% RSLogix 500 project second_Version.RSS, saved by version 8.30.00.16 %
PROJECT "UNTITLED"    % processor: Bul.1763 MicroLogix 1100 Series B %

PROGRAM FILES
  LAD 2   5 rungs
  LAD 3 "CYCLE"  6 rungs
  LAD 4 "ALARMS"  9 rungs
  LAD 5 "IO"  13 rungs
  LAD 6 "LOGIC"  5 rungs

DATA FILES
  O0 OUTPUT  4 elements
  I1 INPUT  6 elements
  S2 STATUS  66 elements
  B3 BINARY  6 elements
  T4 TIMER  4 elements
  C5 COUNTER  1 elements
  R6 CONTROL  1 elements
  N7 INTEGER  4 elements
  F8 FLOAT  1 elements

LADDER 2
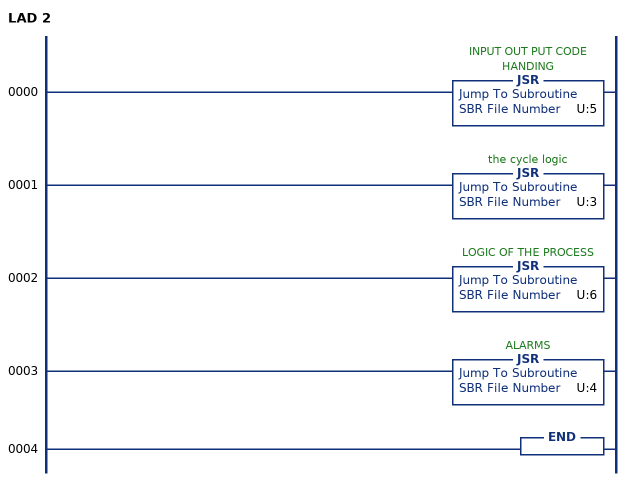
% Rung: 0 %
SOR JSR U:5 EOR
%   U:5  "INPUT OUT PUT CODE HANDING" %
% Rung: 1 %
SOR JSR U:3 EOR
%   U:3  "the cycle logic" %
% Rung: 2 %
SOR JSR U:6 EOR
%   U:6  "LOGIC OF THE PROCESS" %
% Rung: 3 %
SOR JSR U:4 EOR
%   U:4  "ALARMS" %
% Rung: 4 %
SOR END EOR

LADDER 3 "CYCLE"
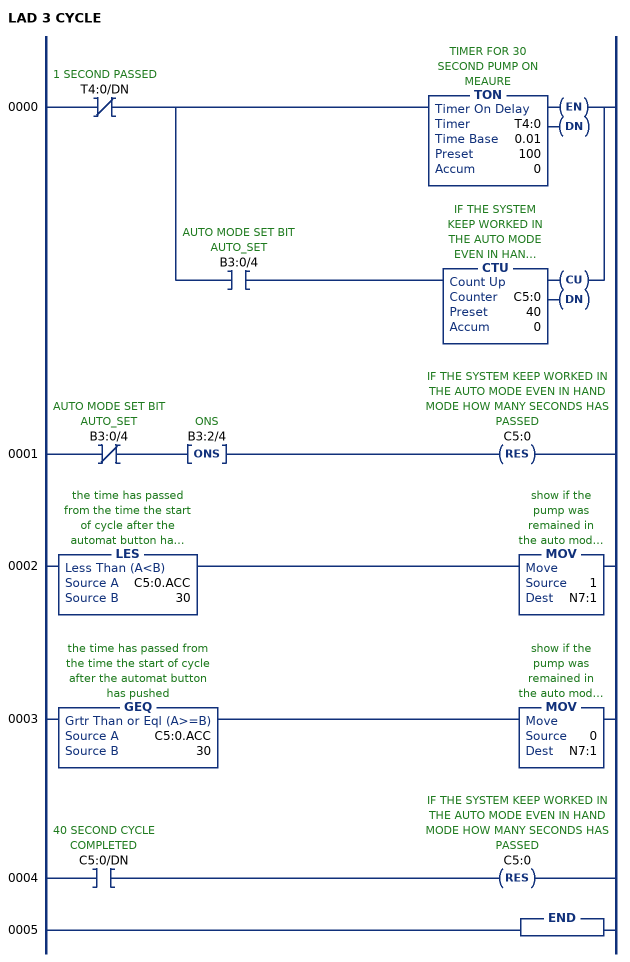
% Rung: 0 %
SOR XIO T4:0/DN BST TON T4:0 0.01 100 0 NXB XIC B3:0/4 CTU C5:0 40 0 BND EOR
%   T4:0/DN  "1 SECOND PASSED" %
%   T4:0  "TIMER FOR 30 SECOND PUMP ON MEAURE" %
%   B3:0/4  AUTO_SET  "AUTO MODE SET BIT" %
%   C5:0  "IF THE SYSTEM KEEP WORKED IN THE AUTO MODE EVEN IN HAND MODE HOW MANY SECONDS HAS PASSED" %
% Rung: 1 %
SOR XIO B3:0/4 ONS B3:2/4 RES C5:0 EOR
%   B3:0/4  AUTO_SET  "AUTO MODE SET BIT" %
%   B3:2/4  "ONS" %
%   C5:0  "IF THE SYSTEM KEEP WORKED IN THE AUTO MODE EVEN IN HAND MODE HOW MANY SECONDS HAS PASSED" %
% Rung: 2 %
SOR LES C5:0.ACC 30 MOV 1 N7:1 EOR
%   C5:0.ACC  "the time has passed from the time the start of cycle after the automat button has pushed" %
%   N7:1  MODE_REF  "show if the pump was remained in the auto mode it should be on which part 1= on mode 0 = off" %
% Rung: 3 %
SOR GEQ C5:0.ACC 30 MOV 0 N7:1 EOR
%   C5:0.ACC  "the time has passed from the time the start of cycle after the automat button has pushed" %
%   N7:1  MODE_REF  "show if the pump was remained in the auto mode it should be on which part 1= on mode 0 = off" %
% Rung: 4 %
SOR XIC C5:0/DN RES C5:0 EOR
%   C5:0/DN  "40 SECOND CYCLE COMPLETED" %
%   C5:0  "IF THE SYSTEM KEEP WORKED IN THE AUTO MODE EVEN IN HAND MODE HOW MANY SECONDS HAS PASSED" %
% Rung: 5 %
SOR END EOR

LADDER 4 "ALARMS"
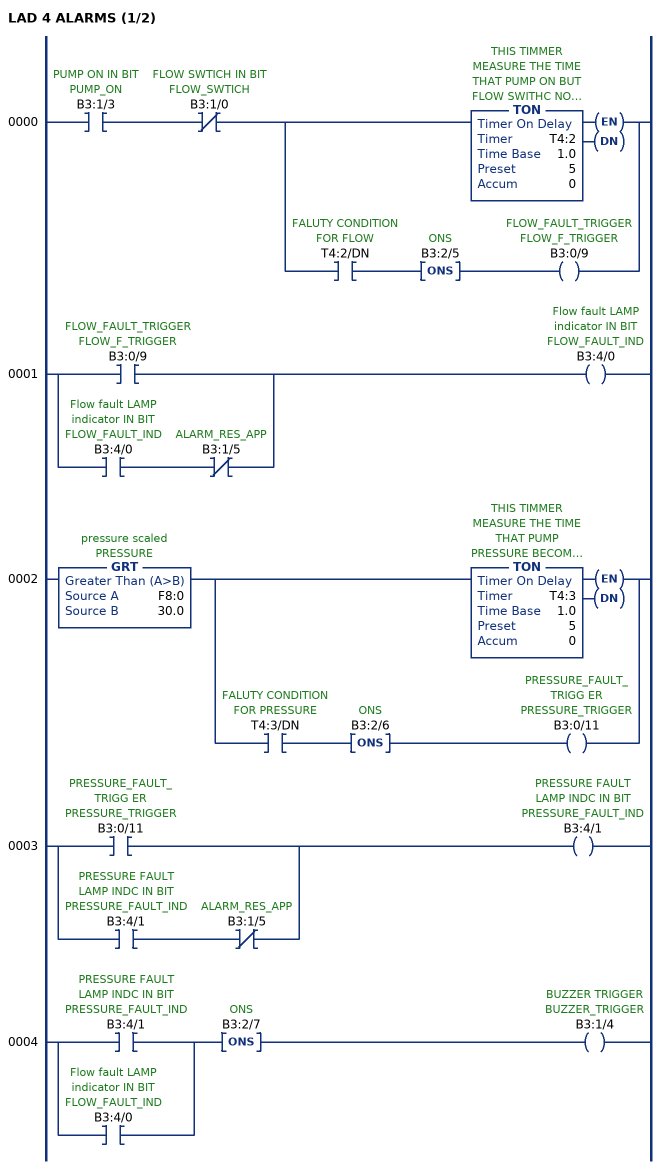
% Rung: 0 %
SOR XIC B3:1/3 XIO B3:1/0 BST TON T4:2 1.0 5 0 NXB XIC T4:2/DN ONS B3:2/5 OTE B3:0/9 BND EOR
%   B3:1/3  PUMP_ON  "PUMP ON IN BIT" %
%   B3:1/0  FLOW_SWTICH  "FLOW SWTICH IN BIT" %
%   T4:2  FLOW_AL_TIM  "THIS TIMMER MEASURE THE TIME THAT PUMP ON BUT FLOW SWITHC NOT TURN ON" %
%   T4:2/DN  "FALUTY CONDITION FOR FLOW" %
%   B3:2/5  "ONS" %
%   B3:0/9  FLOW_F_TRIGGER  "FLOW_FAULT_TRIGGER" %
% Rung: 1 %
SOR BST XIC B3:0/9 NXB XIC B3:4/0 XIO B3:1/5 BND OTE B3:4/0 EOR
%   B3:0/9  FLOW_F_TRIGGER  "FLOW_FAULT_TRIGGER" %
%   B3:4/0  FLOW_FAULT_IND  "Flow fault LAMP indicator IN BIT" %
%   B3:1/5  ALARM_RES_APP %
% Rung: 2 %
SOR GRT F8:0 30.0 BST TON T4:3 1.0 5 0 NXB XIC T4:3/DN ONS B3:2/6 OTE B3:0/11 BND EOR
%   F8:0  PRESSURE  "pressure scaled" %
%   T4:3  PRESSURE_AL_TIM  "THIS TIMMER MEASURE THE TIME THAT PUMP PRESSURE BECOME MORE THAN 30 PSI" %
%   T4:3/DN  "FALUTY CONDITION FOR PRESSURE" %
%   B3:2/6  "ONS" %
%   B3:0/11  PRESSURE_TRIGGER  "PRESSURE_FAULT_TRIGG ER" %
% Rung: 3 %
SOR BST XIC B3:0/11 NXB XIC B3:4/1 XIO B3:1/5 BND OTE B3:4/1 EOR
%   B3:0/11  PRESSURE_TRIGGER  "PRESSURE_FAULT_TRIGG ER" %
%   B3:4/1  PRESSURE_FAULT_IND  "PRESSURE FAULT LAMP INDC IN BIT" %
%   B3:1/5  ALARM_RES_APP %
% Rung: 4 %
SOR BST XIC B3:4/1 NXB XIC B3:4/0 BND ONS B3:2/7 OTE B3:1/4 EOR
%   B3:4/1  PRESSURE_FAULT_IND  "PRESSURE FAULT LAMP INDC IN BIT" %
%   B3:4/0  FLOW_FAULT_IND  "Flow fault LAMP indicator IN BIT" %
%   B3:2/7  "ONS" %
%   B3:1/4  BUZZER_TRIGGER  "BUZZER TRIGGER" %

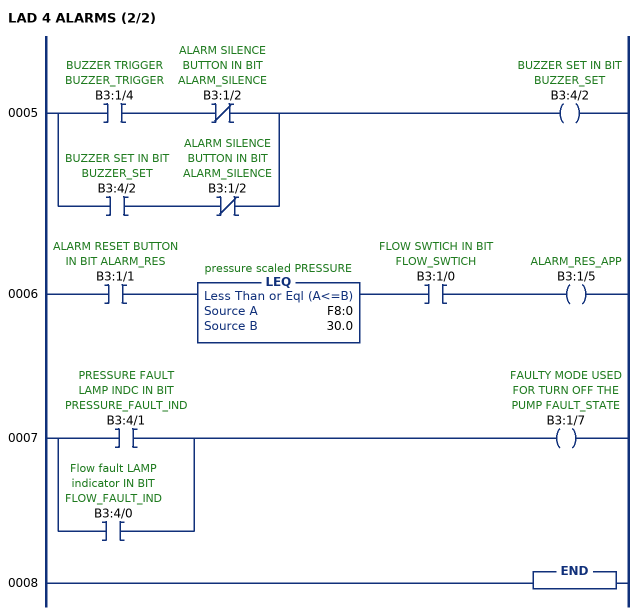
% Rung: 5 %
SOR BST XIC B3:1/4 XIO B3:1/2 NXB XIC B3:4/2 XIO B3:1/2 BND OTE B3:4/2 EOR
%   B3:1/4  BUZZER_TRIGGER  "BUZZER TRIGGER" %
%   B3:1/2  ALARM_SILENCE  "ALARM SILENCE BUTTON IN BIT" %
%   B3:4/2  BUZZER_SET  "BUZZER SET IN BIT" %
% Rung: 6 %
SOR XIC B3:1/1 LEQ F8:0 30.0 XIC B3:1/0 OTE B3:1/5 EOR
%   B3:1/1  ALARM_RES  "ALARM RESET BUTTON IN BIT" %
%   F8:0  PRESSURE  "pressure scaled" %
%   B3:1/0  FLOW_SWTICH  "FLOW SWTICH IN BIT" %
%   B3:1/5  ALARM_RES_APP %
% Rung: 7 %
SOR BST XIC B3:4/1 NXB XIC B3:4/0 BND OTE B3:1/7 EOR
%   B3:4/1  PRESSURE_FAULT_IND  "PRESSURE FAULT LAMP INDC IN BIT" %
%   B3:4/0  FLOW_FAULT_IND  "Flow fault LAMP indicator IN BIT" %
%   B3:1/7  FAULT_STATE  "FAULTY MODE USED FOR TURN OFF THE PUMP" %
% Rung: 8 %
SOR END EOR

LADDER 5 "IO"
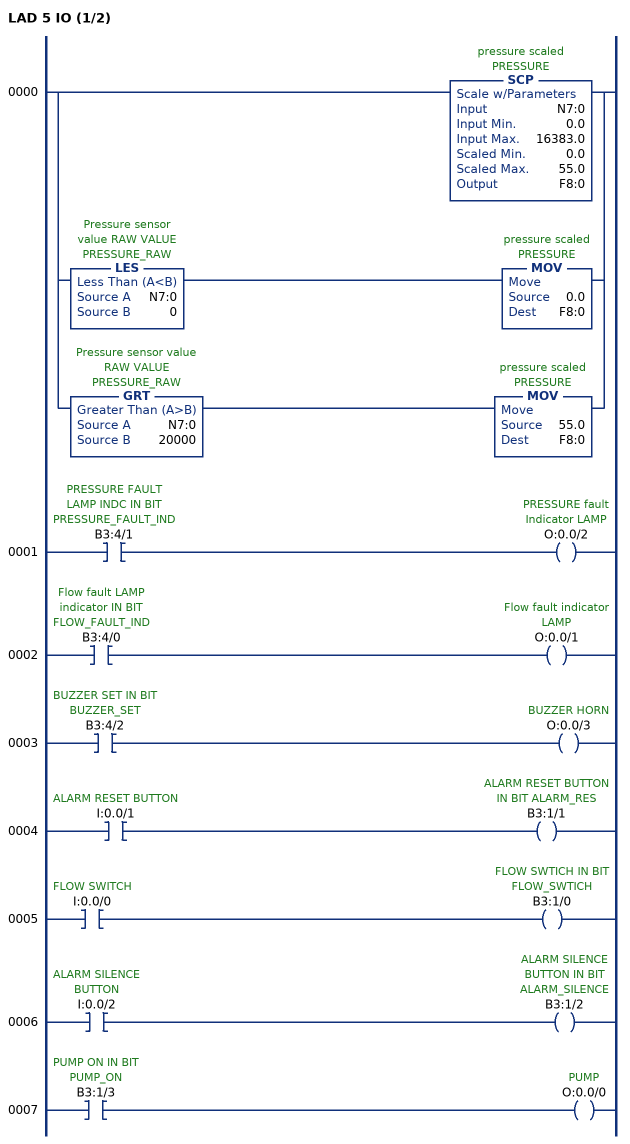
% Rung: 0 %
SOR BST SCP N7:0 0.0 16383.0 0.0 55.0 F8:0 NXB BST LES N7:0 0 MOV 0.0 F8:0 NXB GRT N7:0 20000 MOV 55.0 F8:0 BND BND EOR
%   N7:0  PRESSURE_RAW  "Pressure sensor value RAW VALUE" %
%   F8:0  PRESSURE  "pressure scaled" %
% Rung: 1 %
SOR XIC B3:4/1 OTE O:0.0/2 EOR
%   B3:4/1  PRESSURE_FAULT_IND  "PRESSURE FAULT LAMP INDC IN BIT" %
%   O:0.0/2  "PRESSURE fault Indicator LAMP" %
% Rung: 2 %
SOR XIC B3:4/0 OTE O:0.0/1 EOR
%   B3:4/0  FLOW_FAULT_IND  "Flow fault LAMP indicator IN BIT" %
%   O:0.0/1  "Flow fault indicator LAMP" %
% Rung: 3 %
SOR XIC B3:4/2 OTE O:0.0/3 EOR
%   B3:4/2  BUZZER_SET  "BUZZER SET IN BIT" %
%   O:0.0/3  "BUZZER HORN" %
% Rung: 4 %
SOR XIC I:0.0/1 OTE B3:1/1 EOR
%   I:0.0/1  "ALARM RESET BUTTON" %
%   B3:1/1  ALARM_RES  "ALARM RESET BUTTON IN BIT" %
% Rung: 5 %
SOR XIC I:0.0/0 OTE B3:1/0 EOR
%   I:0.0/0  "FLOW SWITCH" %
%   B3:1/0  FLOW_SWTICH  "FLOW SWTICH IN BIT" %
% Rung: 6 %
SOR XIC I:0.0/2 OTE B3:1/2 EOR
%   I:0.0/2  "ALARM SILENCE BUTTON" %
%   B3:1/2  ALARM_SILENCE  "ALARM SILENCE BUTTON IN BIT" %
% Rung: 7 %
SOR XIC B3:1/3 OTE O:0.0/0 EOR
%   B3:1/3  PUMP_ON  "PUMP ON IN BIT" %
%   O:0.0/0  "PUMP" %

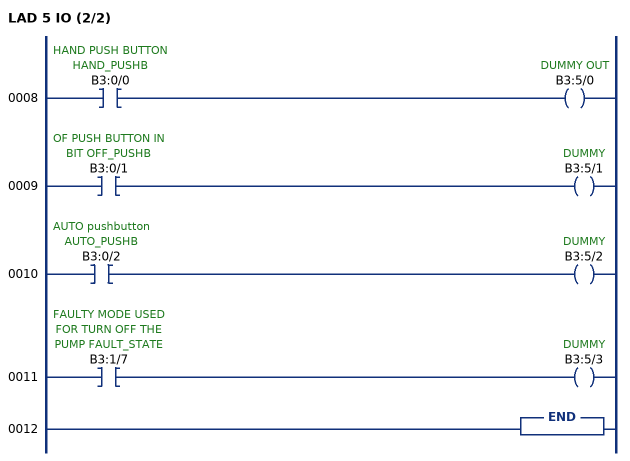
% Rung: 8 %
SOR XIC B3:0/0 OTE B3:5/0 EOR
%   B3:0/0  HAND_PUSHB  "HAND PUSH BUTTON" %
%   B3:5/0  "DUMMY OUT" %
% Rung: 9 %
SOR XIC B3:0/1 OTE B3:5/1 EOR
%   B3:0/1  OFF_PUSHB  "OF PUSH BUTTON IN BIT" %
%   B3:5/1  "DUMMY" %
% Rung: 10 %
SOR XIC B3:0/2 OTE B3:5/2 EOR
%   B3:0/2  AUTO_PUSHB  "AUTO pushbutton" %
%   B3:5/2  "DUMMY" %
% Rung: 11 %
SOR XIC B3:1/7 OTE B3:5/3 EOR
%   B3:1/7  FAULT_STATE  "FAULTY MODE USED FOR TURN OFF THE PUMP" %
%   B3:5/3  "DUMMY" %
% Rung: 12 %
SOR END EOR

LADDER 6 "LOGIC"
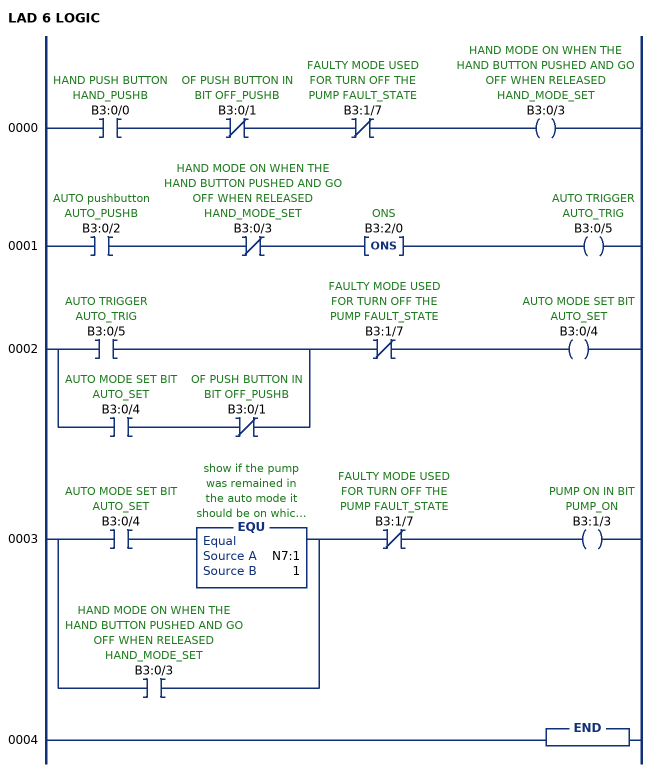
% Rung: 0 %
SOR XIC B3:0/0 XIO B3:0/1 XIO B3:1/7 OTE B3:0/3 EOR
%   B3:0/0  HAND_PUSHB  "HAND PUSH BUTTON" %
%   B3:0/1  OFF_PUSHB  "OF PUSH BUTTON IN BIT" %
%   B3:1/7  FAULT_STATE  "FAULTY MODE USED FOR TURN OFF THE PUMP" %
%   B3:0/3  HAND_MODE_SET  "HAND MODE ON WHEN THE HAND BUTTON PUSHED AND GO OFF WHEN RELEASED" %
% Rung: 1 %
SOR XIC B3:0/2 XIO B3:0/3 ONS B3:2/0 OTE B3:0/5 EOR
%   B3:0/2  AUTO_PUSHB  "AUTO pushbutton" %
%   B3:0/3  HAND_MODE_SET  "HAND MODE ON WHEN THE HAND BUTTON PUSHED AND GO OFF WHEN RELEASED" %
%   B3:2/0  "ONS" %
%   B3:0/5  AUTO_TRIG  "AUTO TRIGGER" %
% Rung: 2 %
SOR BST XIC B3:0/5 NXB XIC B3:0/4 XIO B3:0/1 BND XIO B3:1/7 OTE B3:0/4 EOR
%   B3:0/5  AUTO_TRIG  "AUTO TRIGGER" %
%   B3:0/4  AUTO_SET  "AUTO MODE SET BIT" %
%   B3:0/1  OFF_PUSHB  "OF PUSH BUTTON IN BIT" %
%   B3:1/7  FAULT_STATE  "FAULTY MODE USED FOR TURN OFF THE PUMP" %
% Rung: 3 %
SOR BST XIC B3:0/4 EQU N7:1 1 NXB XIC B3:0/3 BND XIO B3:1/7 OTE B3:1/3 EOR
%   B3:0/4  AUTO_SET  "AUTO MODE SET BIT" %
%   N7:1  MODE_REF  "show if the pump was remained in the auto mode it should be on which part 1= on mode 0 = off" %
%   B3:0/3  HAND_MODE_SET  "HAND MODE ON WHEN THE HAND BUTTON PUSHED AND GO OFF WHEN RELEASED" %
%   B3:1/7  FAULT_STATE  "FAULTY MODE USED FOR TURN OFF THE PUMP" %
%   B3:1/3  PUMP_ON  "PUMP ON IN BIT" %
% Rung: 4 %
SOR END EOR

OTHER DOCUMENTED ADDRESSES
  B3:0/6  AUTO_INTERUPT  "AUTO INTERUPT"
  B3:0/7  STOPMODE_SET  "stop mode set bit"
  B3:0/8  NOT_AUTOSET_BIT  "this bit Not logic of auto set bit"
  B3:0/10  FLOW_FAULT_SET  "FLOW FAULT SET BIT"
  B3:0/15  "TEST"
  B3:2/1  "ONS"
  N7:2  CURRENT_MODE  "pump current mode hand mode = 2 auto mode = 1 stop mode = 0"
  T4:1  "TIMER FOR MEASRUING THE OFF TIME MOTOR IN AUTOMATE MODE"

REVISION NOTES
  0: “In this simplified logic, the counter always resets whenever AUTO is selected, regardless of whether the previous mode was OFF or HAND, making the program clearer but less realistic

DATA TABLE (non-zero values as saved)
DATA T4
% .PRE .ACC %
% T4:0 % 100 0
% T4:2 % 5 0
% T4:3 % 5 0
DATA C5
% .PRE .ACC %
% C5:0 % 40 0
